(* CODESYS project Brauanlagev3.project

Project tree, tasks and I/O mapping:
  Device : CODESYS Control for Raspberry Pi, 3S - Smart Software Solutions GmbH, version 3.5.9.20
    application Application
      libraries: Standard, * (System); SysProcess, 3.5.7.0 (System); VisuDialogs, * (System); BASIC, 3.3.3.0 (OSCAT); SysTypes Interfaces, * (System); SysMem, 3.5.5.0 (System)
      task VISU_TASK (cyclic, interval 100 ms, priority 31) calls VisuElems.Visu_Prg
      task LinuxSystemTask (cyclic, interval 1000 ms, priority 31) calls RPI_SYSTEM
      task IO (cyclic, interval 10 ms, priority 1) calls IOCOM
      task KI (cyclic, interval 10 ms, priority 1) calls Automatik
      global variables Variablenliste
      visualisation Visualization
      program Automatik [ST]
      visualisation Setup
      visualisation Settings
      program IOCOM [ST]
      program RPI_SYSTEM [ST]
      global variables PersistentVars
    SoftMotion General Axis Pool
    I²C
    SPI
    GPIOs_B_Pi2 : GPIOs B+/Pi2, 3S - Smart Software Solutions GmbH, version 1.1.1.10
        unmapped channels: digital inputs (GPIO0..GPIO31), digital outputs (GPIO0..GPIO31)
    Onewire
      Onewire_master : Onewire master, 3S - Smart Software Solutions GmbH, version 1.0.0.0
        DS18B20 : DS18B20, 3S - Smart Software Solutions GmbH, version 1.3.0.0
            settings: Unique device address = '28-011572667aff'
        DS18B20_2 : DS18B20, 3S - Smart Software Solutions GmbH, version 1.3.0.0
            settings: Unique device address = '28-0115726f14ff'
        DS18B20_1 : DS18B20, 3S - Smart Software Solutions GmbH, version 1.3.0.0
            settings: Unique device address = '28-0115729769ff'
    Camera device
      <Leer>
  libraries: VisuSymbols, 3.5.8.0 (System)
  text list GlobalTextList
  text list System
*)

// Device/Application/Variablenliste
VAR_GLOBAL
	AUTO_VERBLEIBENDE_ZEIT:TIME;
	seek:UINT;
	seek2:UINT;
	IN_TEMP_1:REAL:=0;
	IN_TEMP_2:REAL:=0;
	IN_TEMP_3:REAL:=0;
	OUT_TOPF_2_ON:BOOL:=0;
	OUT_220_1_ON:BOOL:=0;
	OUT_220_2_ON:BOOL:=0;
	OUT_24_1_ON:BOOL:=0;
	OUT_24_2_ON:BOOL:=0;
	OUT_DOSE_1_ON:BOOL:=0;
	OUT_DOSE_2_ON:BOOL:=0;
	OUT_DOSE_3_ON:BOOL:=0;
	OUT_DOSE_4_ON:BOOL:=0;
	OUT_ALARM_ON:BOOL:=0;
END_VAR

{attribute 'qualified_only'}
VAR_GLOBAL PERSISTENT RETAIN
	// Laufzeitvariablen
	AUTO_ZYKLUS:UINT;
	AUTO_REZEPT:UINT;
	AUTO_ON:BOOL;
	// Automatik Rezept
	SET_AUTO_REZEPT_NAME:ARRAY[0..100] OF STRING;
	SET_AUTO_NAME:ARRAY[0..100,0..100] OF STRING;
	SET_AUTO_ZEIT:ARRAY[0..100,0..100] OF UINT;
	SET_AUTO_TIMER_ON:ARRAY[0..100,0..100] OF BOOL;
	SET_AUTO_ALARM:ARRAY[0..100,0..100] OF BOOL;	
	SET_AUTO_TOPF_1_ON:ARRAY[0..100,0..100] OF BOOL;
	SET_AUTO_TOPF_3_ON:ARRAY[0..100,0..100] OF BOOL;
	SET_AUTO_TOPF_1_TARGET:ARRAY[0..100,0..100] OF REAL;
	SET_AUTO_TOPF_3_TARGET:ARRAY[0..100,0..100] OF REAL;
	SET_AUTO_DOSE_1_ON:ARRAY[0..100,0..100] OF BOOL;
	SET_AUTO_DOSE_2_ON:ARRAY[0..100,0..100] OF BOOL;	
	SET_AUTO_DOSE_3_ON:ARRAY[0..100,0..100] OF BOOL;	
	SET_AUTO_DOSE_4_ON:ARRAY[0..100,0..100] OF BOOL;
	// Einstellungen
	SET_TOPF_1_AUTO:BOOL;
	SET_TOPF_3_AUTO:BOOL;
	SET_TOPF_1_TARGET:REAL;
	SET_TOPF_3_TARGET:REAL;
	SET_TOPF_1_HYSTERESIS:REAL:=2;
	SET_TOPF_3_HYSTERESIS:REAL:=2;
	SET_TOPF_1_HYSTERESIS2:REAL:=2;
	SET_TOPF_3_HYSTERESIS2:REAL:=2;
	SET_TOPF_1_ON:BOOL;
	SET_TOPF_3_ON:BOOL;
	SET_TOPF_1_NAME:STRING:='TOPF1';
	SET_TOPF_2_NAME:STRING:='TOPF2';
	SET_TOPF_3_NAME:STRING:='TOPF3';
	SET_DOSE_1_AUTO:BOOL;
	SET_DOSE_2_AUTO:BOOL;
	SET_DOSE_3_AUTO:BOOL;
	SET_DOSE_4_AUTO:BOOL;
	SET_DOSE_1_NAME:STRING:='DOSE1';
	SET_DOSE_2_NAME:STRING:='DOSE2';
	SET_DOSE_3_NAME:STRING:='DOSE3';
	SET_DOSE_4_NAME:STRING:='DOSE4';
END_VAR

// Device/Application/PersistentVars
{attribute 'qualified_only'}
VAR_GLOBAL PERSISTENT RETAIN

	// Instanzpfad der persistenten Variablen erzeugt
	Variablenliste.AUTO_ZYKLUS: UINT;
	// Instanzpfad der persistenten Variablen erzeugt
	Variablenliste.AUTO_REZEPT: UINT;
	// Instanzpfad der persistenten Variablen erzeugt
	Variablenliste.AUTO_ON: BOOL;
	// Instanzpfad der persistenten Variablen erzeugt
	Variablenliste.SET_AUTO_REZEPT_NAME: ARRAY [0..100] OF STRING;
	// Instanzpfad der persistenten Variablen erzeugt
	Variablenliste.SET_AUTO_NAME: ARRAY [0..100, 0..100] OF STRING;
	// Instanzpfad der persistenten Variablen erzeugt
	Variablenliste.SET_AUTO_ZEIT: ARRAY [0..100, 0..100] OF UINT;
	// Instanzpfad der persistenten Variablen erzeugt
	Variablenliste.SET_AUTO_TIMER_ON: ARRAY [0..100, 0..100] OF BOOL;
	// Instanzpfad der persistenten Variablen erzeugt
	Variablenliste.SET_AUTO_ALARM: ARRAY [0..100, 0..100] OF BOOL;
	// Instanzpfad der persistenten Variablen erzeugt
	Variablenliste.SET_AUTO_TOPF_1_ON: ARRAY [0..100, 0..100] OF BOOL;
	// Instanzpfad der persistenten Variablen erzeugt
	Variablenliste.SET_AUTO_TOPF_3_ON: ARRAY [0..100, 0..100] OF BOOL;
	// Instanzpfad der persistenten Variablen erzeugt
	Variablenliste.SET_AUTO_TOPF_1_TARGET: ARRAY [0..100, 0..100] OF REAL;
	// Instanzpfad der persistenten Variablen erzeugt
	Variablenliste.SET_AUTO_TOPF_3_TARGET: ARRAY [0..100, 0..100] OF REAL;
	// Instanzpfad der persistenten Variablen erzeugt
	Variablenliste.SET_AUTO_DOSE_1_ON: ARRAY [0..100, 0..100] OF BOOL;
	// Instanzpfad der persistenten Variablen erzeugt
	Variablenliste.SET_AUTO_DOSE_2_ON: ARRAY [0..100, 0..100] OF BOOL;
	// Instanzpfad der persistenten Variablen erzeugt
	Variablenliste.SET_AUTO_DOSE_3_ON: ARRAY [0..100, 0..100] OF BOOL;
	// Instanzpfad der persistenten Variablen erzeugt
	Variablenliste.SET_AUTO_DOSE_4_ON: ARRAY [0..100, 0..100] OF BOOL;
	// Instanzpfad der persistenten Variablen erzeugt
	Variablenliste.SET_TOPF_1_AUTO: BOOL;
	// Instanzpfad der persistenten Variablen erzeugt
	Variablenliste.SET_TOPF_3_AUTO: BOOL;
	// Instanzpfad der persistenten Variablen erzeugt
	Variablenliste.SET_TOPF_1_TARGET: REAL;
	// Instanzpfad der persistenten Variablen erzeugt
	Variablenliste.SET_TOPF_3_TARGET: REAL;
	// Instanzpfad der persistenten Variablen erzeugt
	Variablenliste.SET_TOPF_1_HYSTERESIS: REAL := 2.0;
	// Instanzpfad der persistenten Variablen erzeugt
	Variablenliste.SET_TOPF_3_HYSTERESIS: REAL := 2.0;
	// Instanzpfad der persistenten Variablen erzeugt
	Variablenliste.SET_TOPF_1_HYSTERESIS2: REAL := 2.0;
	// Instanzpfad der persistenten Variablen erzeugt
	Variablenliste.SET_TOPF_3_HYSTERESIS2: REAL := 2.0;
	// Instanzpfad der persistenten Variablen erzeugt
	Variablenliste.SET_TOPF_1_ON: BOOL;
	// Instanzpfad der persistenten Variablen erzeugt
	Variablenliste.SET_TOPF_3_ON: BOOL;
	// Instanzpfad der persistenten Variablen erzeugt
	Variablenliste.SET_TOPF_1_NAME: STRING := 'TOPF1';
	// Instanzpfad der persistenten Variablen erzeugt
	Variablenliste.SET_TOPF_2_NAME: STRING := 'TOPF2';
	// Instanzpfad der persistenten Variablen erzeugt
	Variablenliste.SET_TOPF_3_NAME: STRING := 'TOPF3';
	// Instanzpfad der persistenten Variablen erzeugt
	Variablenliste.SET_DOSE_1_AUTO: BOOL;
	// Instanzpfad der persistenten Variablen erzeugt
	Variablenliste.SET_DOSE_2_AUTO: BOOL;
	// Instanzpfad der persistenten Variablen erzeugt
	Variablenliste.SET_DOSE_3_AUTO: BOOL;
	// Instanzpfad der persistenten Variablen erzeugt
	Variablenliste.SET_DOSE_4_AUTO: BOOL;
	// Instanzpfad der persistenten Variablen erzeugt
	Variablenliste.SET_DOSE_1_NAME: STRING := 'DOSE1';
	// Instanzpfad der persistenten Variablen erzeugt
	Variablenliste.SET_DOSE_2_NAME: STRING := 'DOSE2';
	// Instanzpfad der persistenten Variablen erzeugt
	Variablenliste.SET_DOSE_3_NAME: STRING := 'DOSE3';
	// Instanzpfad der persistenten Variablen erzeugt
	Variablenliste.SET_DOSE_4_NAME: STRING := 'DOSE4';
END_VAR

// Device/Application/RPI_SYSTEM
PROGRAM RPI_SYSTEM
VAR
   cmdResult   :    RTS_IEC_result;
END_VAR

IF OUT_ALARM_ON THEN 
	// SysProcessExecuteCommand('aplay /media/shared/alarm.wav', ADR(cmdResult)); 
	// SysProcessExecuteCommand('python /media/shared/alarm.py', ADR(cmdResult)); 
END_IF

END_PROGRAM

// Device/Application/IOCOM
PROGRAM IOCOM
VAR
	rTemp: REAL;
END_VAR


%QX0.5:=NOT OUT_DOSE_1_ON;
%QX0.6:=NOT OUT_DOSE_2_ON;
%QX1.4:=NOT OUT_DOSE_3_ON;
%QX1.5:=NOT OUT_DOSE_4_ON;
%QX2.0:=NOT OUT_220_1_ON;
%QX2.3:=NOT OUT_220_2_ON;
%QX2.4:=NOT OUT_24_1_ON;
%QX2.5:=NOT OUT_24_2_ON;
IN_TEMP_1:=DS18B20.rTemp;
IN_TEMP_2:=DS18b20_1.rTemp;
IN_TEMP_3:=DS18b20_2.rTemp;

END_PROGRAM

// Device/Application/Automatik
PROGRAM Automatik
VAR
	TIMER:TON;
END_VAR

(*TODO
ALARM pwm jack`?
*)


TIMER(IN:=SET_AUTO_TIMER_ON[AUTO_ZYKLUS,AUTO_REZEPT] AND AUTO_ON AND NOT TIMER.Q, PT:=LWORD_TO_TIME(UINT_TO_LWORD(SET_AUTO_ZEIT[AUTO_ZYKLUS,AUTO_REZEPT])*60000));
(*TIMER.ET:=ELAPSED;*)
AUTO_VERBLEIBENDE_ZEIT:=LWORD_TO_TIME(UINT_TO_LWORD(SET_AUTO_ZEIT[AUTO_ZYKLUS,AUTO_REZEPT])*60000)-TIMER.ET;


IF TIMER.Q THEN
	AUTO_ZYKLUS:=AUTO_ZYKLUS+1;
	IF SET_AUTO_ALARM[AUTO_ZYKLUS,AUTO_REZEPT] THEN
		OUT_ALARM_ON:=TRUE;
	END_IF
END_IF



IF AUTO_ON THEN
	IF SET_DOSE_1_AUTO THEN
		IF SET_AUTO_DOSE_1_ON[AUTO_ZYKLUS,AUTO_REZEPT] THEN
			OUT_DOSE_1_ON:=TRUE;
		ELSE 
			OUT_DOSE_1_ON:=FALSE;
		END_IF
	END_IF
	
	IF SET_DOSE_2_AUTO THEN
		IF SET_AUTO_DOSE_2_ON[AUTO_ZYKLUS,AUTO_REZEPT] THEN
			OUT_DOSE_2_ON:=TRUE;
		ELSE 
			OUT_DOSE_2_ON:=FALSE;
		END_IF
	END_IF

	IF SET_DOSE_3_AUTO THEN
		IF SET_AUTO_DOSE_3_ON[AUTO_ZYKLUS,AUTO_REZEPT] THEN
			OUT_DOSE_3_ON:=TRUE;
		ELSE 
			OUT_DOSE_3_ON:=FALSE;
		END_IF
	END_IF

	IF SET_DOSE_4_AUTO THEN
		IF SET_AUTO_DOSE_4_ON[AUTO_ZYKLUS,AUTO_REZEPT] THEN
			OUT_DOSE_4_ON:=TRUE;
		ELSE 
			OUT_DOSE_4_ON:=FALSE;
		END_IF
	END_IF

	IF SET_TOPF_1_AUTO THEN
		IF SET_AUTO_TOPF_1_ON[AUTO_ZYKLUS,AUTO_REZEPT] THEN
			SET_TOPF_1_TARGET:=SET_AUTO_TOPF_1_TARGET[AUTO_ZYKLUS,AUTO_REZEPT];
			SET_TOPF_1_ON:=TRUE;
		ELSE
			SET_TOPF_1_ON:=FALSE;
		END_IF
	END_IF

	IF SET_TOPF_3_AUTO THEN
		IF SET_AUTO_TOPF_3_ON[AUTO_ZYKLUS,AUTO_REZEPT] THEN
			SET_TOPF_3_TARGET:=SET_AUTO_TOPF_3_TARGET[AUTO_ZYKLUS,AUTO_REZEPT];
			SET_TOPF_3_ON:=TRUE;
		ELSE
			SET_TOPF_3_ON:=FALSE;
		END_IF
	END_IF
END_IF

IF SET_TOPF_1_ON THEN
	IF IN_TEMP_1 > SET_TOPF_1_TARGET THEN
		OUT_220_1_ON:=FALSE;
		OUT_24_1_ON:=FALSE;
	END_IF
	IF IN_TEMP_1 < SET_TOPF_1_TARGET - SET_TOPF_1_HYSTERESIS THEN
		OUT_220_1_ON:=TRUE;
	END_IF
	IF IN_TEMP_1 < SET_TOPF_1_TARGET - SET_TOPF_1_HYSTERESIS - SET_TOPF_1_HYSTERESIS2 THEN
		OUT_24_1_ON:=TRUE;
	ELSE
		OUT_24_1_ON:=FALSE;
	END_IF
ELSE 
	OUT_220_1_ON:=FALSE;
	OUT_24_1_ON:=FALSE;
END_IF

IF SET_TOPF_3_ON THEN
	IF IN_TEMP_3 > SET_TOPF_3_TARGET THEN
		OUT_220_2_ON:=FALSE;
		OUT_24_2_ON:=FALSE;
	END_IF
	IF IN_TEMP_3 < SET_TOPF_3_TARGET - SET_TOPF_3_HYSTERESIS THEN
		OUT_220_2_ON:=TRUE;
	END_IF
	IF IN_TEMP_3 < SET_TOPF_3_TARGET - SET_TOPF_3_HYSTERESIS - SET_TOPF_3_HYSTERESIS2 THEN
		OUT_24_2_ON:=TRUE;
	ELSE
		OUT_24_2_ON:=FALSE;
	END_IF
ELSE 
	OUT_220_2_ON:=FALSE;
	OUT_24_2_ON:=FALSE;
END_IF

END_PROGRAM

// Device/Application/Visualization
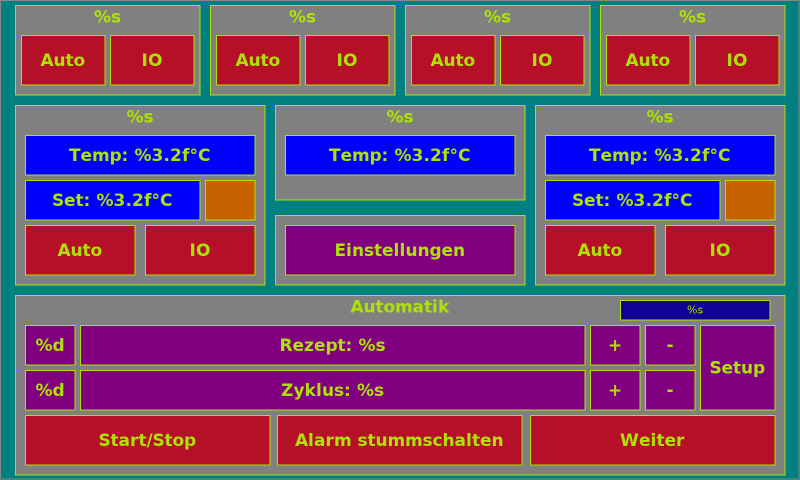
VISUALIZATION Visualization  // 800x480
    RoundedRectangle (15,295 770x180), "Automatik"
    RoundedRectangle (25,415 245x50), "Start/Stop", colour toggle: AUTO_ON
        toggle AUTO_ON
    RoundedRectangle (277,415 245x50), "Alarm stummschalten", colour toggle: OUT_ALARM_ON
        OnMouseDown: execute { OUT_ALARM_ON:=0; }
    RoundedRectangle (700,325 75x85), "Setup"
        OnMouseDown:  Assign=Setup, Type=Assignment
    RoundedRectangle (530,415 245x50), "Weiter"
        OnMouseDown: execute { AUTO_ZYKLUS:=AUTO_ZYKLUS+1; }
    RoundedRectangle (15,5 185x90), "%s", text variable: SET_DOSE_1_NAME
        OnMouseDown: write the text variable via Edit
    RoundedRectangle (110,35 84x50), "IO", colour toggle: OUT_DOSE_1_ON
        toggle OUT_DOSE_1_ON
    RoundedRectangle (21,35 84x50), "Auto", colour toggle: SET_DOSE_1_AUTO
        toggle SET_DOSE_1_AUTO
    RoundedRectangle (210,5 185x90), "%s", text variable: SET_DOSE_2_NAME
        OnMouseDown: write the text variable via Edit
    RoundedRectangle (305,35 84x50), "IO", colour toggle: OUT_DOSE_2_ON
        toggle OUT_DOSE_2_ON
    RoundedRectangle (216,35 84x50), "Auto", colour toggle: SET_DOSE_2_AUTO
        toggle SET_DOSE_2_AUTO
    RoundedRectangle (405,5 185x90), "%s", text variable: SET_DOSE_3_NAME
        OnMouseDown: write the text variable via Edit
    RoundedRectangle (500,35 84x50), "IO", colour toggle: OUT_DOSE_3_ON
        toggle OUT_DOSE_3_ON
    RoundedRectangle (411,35 84x50), "Auto", colour toggle: SET_DOSE_3_AUTO
        toggle SET_DOSE_3_AUTO
    RoundedRectangle (600,5 185x90), "%s", text variable: SET_DOSE_4_NAME
        OnMouseDown: write the text variable via Edit
    RoundedRectangle (695,35 84x50), "IO", colour toggle: OUT_DOSE_4_ON
        toggle OUT_DOSE_4_ON
    RoundedRectangle (606,35 84x50), "Auto", colour toggle: SET_DOSE_4_AUTO
        toggle SET_DOSE_4_AUTO
    RoundedRectangle (275,105 250x95), "%s", text variable: SET_TOPF_2_NAME
        OnMouseDown: write the text variable via Edit
    RoundedRectangle (285,135 230x40), "Temp: %3.2f°C", text variable: IN_TEMP_2
    RoundedRectangle (535,105 250x180), "%s", text variable: SET_TOPF_3_NAME, colour toggle: OUT_220_2_ON
        OnMouseDown: write the text variable via Edit
    RoundedRectangle (665,225 110x50), "IO", colour toggle: SET_TOPF_3_ON
        toggle SET_TOPF_3_ON
    RoundedRectangle (545,225 110x50), "Auto", colour toggle: SET_TOPF_3_AUTO
        toggle SET_TOPF_3_AUTO
    RoundedRectangle (545,135 230x40), "Temp: %3.2f°C", text variable: IN_TEMP_3
    RoundedRectangle (545,180 175x40), "Set: %3.2f°C", text variable: SET_TOPF_3_TARGET
        OnMouseDown: write the text variable via Edit, min 0, max 105
    RoundedRectangle (725,180 50x40), text variable: SET_TOPF_3_TARGET
        OnMouseDown: write the text variable via VisuDialogs.Numpad, min 0, max 105
    RoundedRectangle (15,105 250x180), "%s", text variable: SET_TOPF_1_NAME, colour toggle: OUT_220_1_ON
        OnMouseDown: write the text variable via Edit
    RoundedRectangle (145,225 110x50), "IO", colour toggle: SET_TOPF_1_ON
        toggle SET_TOPF_1_ON
    RoundedRectangle (25,225 110x50), "Auto", colour toggle: SET_TOPF_1_AUTO
        toggle SET_TOPF_1_AUTO
    RoundedRectangle (25,135 230x40), "Temp: %3.2f°C", text variable: IN_TEMP_1
    RoundedRectangle (25,180 175x40), "Set: %3.2f°C", text variable: SET_TOPF_1_TARGET
        OnMouseDown: write the text variable via Edit, min 0, max 105
    RoundedRectangle (205,180 50x40), text variable: SET_TOPF_1_TARGET
        OnMouseDown: write the text variable via VisuDialogs.Numpad, min 0, max 105
    RoundedRectangle (275,215 250x70)
    RoundedRectangle (285,225 230x50), "Einstellungen"
        OnMouseDown:  Assign=Settings, Type=Assignment
    RoundedRectangle (620,300 150x20), "%s", text variable: AUTO_VERBLEIBENDE_ZEIT, invisible if: NOT SET_AUTO_TIMER_ON[AUTO_ZYKLUS,AUTO_REZEPT]
    RoundedRectangle (590,370 50x40), "+"
        OnMouseDown: execute { AUTO_ZYKLUS:=AUTO_ZYKLUS+1; }
    RoundedRectangle (645,370 50x40), "-"
        OnMouseDown: execute {
            IF AUTO_ZYKLUS > 0 THEN
            	AUTO_ZYKLUS:=AUTO_ZYKLUS-1;
            END_IF;
        }
    RoundedRectangle (80,370 505x40), "Zyklus: %s", text variable: SET_AUTO_NAME[AUTO_ZYKLUS,AUTO_REZEPT]
    RoundedRectangle (25,370 50x40), "%d", text variable: AUTO_ZYKLUS
    RoundedRectangle (590,325 50x40), "+"
        OnMouseDown: execute { AUTO_REZEPT:=AUTO_REZEPT+1; AUTO_ON:=FALSE; }
    RoundedRectangle (645,325 50x40), "-"
        OnMouseDown: execute {
            IF AUTO_REZEPT > 0 THEN
            	AUTO_REZEPT:=AUTO_REZEPT-1;
            END_IF;
            AUTO_ON:=FALSE;
        }
    RoundedRectangle (80,325 505x40), "Rezept: %s", text variable: SET_AUTO_REZEPT_NAME[AUTO_REZEPT]
    RoundedRectangle (25,325 50x40), "%d", text variable: AUTO_REZEPT
END_VISUALIZATION

// Device/Application/Setup
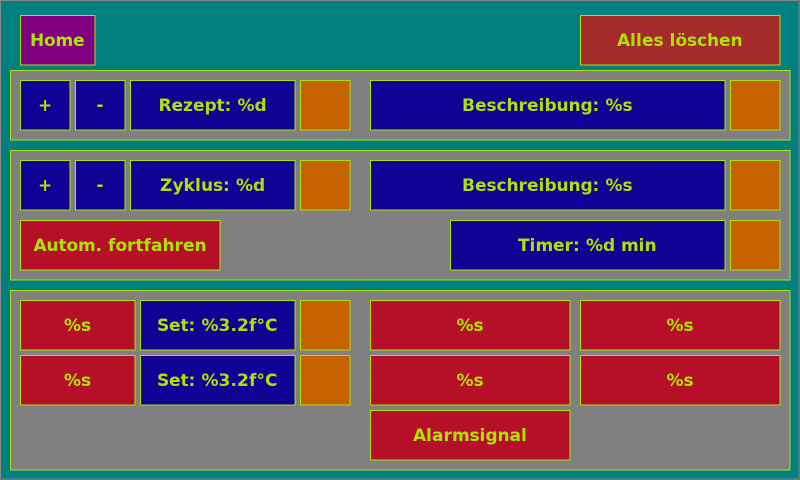
VISUALIZATION Setup  // 800x480
    RoundedRectangle (10,70 780x70)
    RoundedRectangle (10,290 780x180)
    RoundedRectangle (10,150 780x130)
    RoundedRectangle (20,300 115x50), "%s", text variable: SET_TOPF_1_NAME, colour toggle: SET_AUTO_TOPF_1_ON[seek,seek2]
        toggle SET_AUTO_TOPF_1_ON[seek,seek2]
    RoundedRectangle (140,300 155x50), "Set: %3.2f°C", text variable: SET_AUTO_TOPF_1_TARGET[seek,seek2]
        OnMouseDown: write the text variable via Edit
    RoundedRectangle (300,300 50x50), text variable: SET_AUTO_TOPF_1_TARGET[seek,seek2]
        OnMouseDown: write the text variable via VisuDialogs.Numpad
    RoundedRectangle (370,300 200x50), "%s", text variable: SET_DOSE_1_NAME, colour toggle: SET_AUTO_DOSE_1_ON[seek,seek2]
        toggle SET_AUTO_DOSE_1_ON[seek,seek2]
    RoundedRectangle (370,410 200x50), "Alarmsignal", colour toggle: SET_AUTO_ALARM[seek,seek2]
        toggle SET_AUTO_ALARM[seek,seek2]
    RoundedRectangle (20,355 115x50), "%s", text variable: SET_TOPF_3_NAME, colour toggle: SET_AUTO_TOPF_3_ON[seek,seek2]
        toggle SET_AUTO_TOPF_3_ON[seek,seek2]
    RoundedRectangle (300,355 50x50), text variable: SET_AUTO_TOPF_3_TARGET[seek,seek2]
        OnMouseDown: write the text variable via VisuDialogs.Numpad
    RoundedRectangle (140,355 155x50), "Set: %3.2f°C", text variable: SET_AUTO_TOPF_3_TARGET[seek,seek2]
        OnMouseDown: write the text variable via Edit
    RoundedRectangle (370,355 200x50), "%s", text variable: SET_DOSE_2_NAME, colour toggle: SET_AUTO_DOSE_2_ON[seek,seek2]
        toggle SET_AUTO_DOSE_2_ON[seek,seek2]
    RoundedRectangle (580,355 200x50), "%s", text variable: SET_DOSE_4_NAME, colour toggle: SET_AUTO_DOSE_4_ON[seek,seek2]
        toggle SET_AUTO_DOSE_4_ON[seek,seek2]
    RoundedRectangle (580,300 200x50), "%s", text variable: SET_DOSE_3_NAME, colour toggle: SET_AUTO_DOSE_3_ON[seek,seek2]
        toggle SET_AUTO_DOSE_3_ON[seek,seek2]
    RoundedRectangle (20,15 75x50), "Home"
        OnMouseDown:  Assign=Visualization, Type=Assignment
    RoundedRectangle (370,160 355x50), "Beschreibung: %s", text variable: SET_AUTO_NAME[seek,seek2]
        OnMouseDown: write the text variable via Edit
    RoundedRectangle (730,160 50x50), text variable: SET_AUTO_NAME[seek,seek2]
        OnMouseDown: write the text variable via VisuDialogs.Keypad
    RoundedRectangle (20,160 50x50), "+"
        OnMouseDown: execute { seek:=seek+1; }
    RoundedRectangle (75,160 50x50), "-"
        OnMouseDown: execute {
            IF seek > 0 THEN
            	seek:=seek-1;
            END_IF;
        }
    RoundedRectangle (130,160 165x50), "Zyklus: %d", text variable: seek
        OnMouseDown: write the text variable via Edit
    RoundedRectangle (300,160 50x50), text variable: seek
        OnMouseDown: write the text variable via VisuDialogs.Numpad
    RoundedRectangle (450,220 275x50), "Timer: %d min", text variable: SET_AUTO_ZEIT[seek,seek2], invisible if: NOT SET_AUTO_TIMER_ON[seek,seek2]
        OnMouseDown: write the text variable via Edit
    RoundedRectangle (730,220 50x50), text variable: SET_AUTO_ZEIT[seek,seek2], invisible if: NOT SET_AUTO_TIMER_ON[seek,seek2]
        OnMouseDown: write the text variable via VisuDialogs.Numpad
    RoundedRectangle (20,220 200x50), "Autom. fortfahren", colour toggle: SET_AUTO_TIMER_ON[seek,seek2]
        toggle SET_AUTO_TIMER_ON[seek,seek2]
    RoundedRectangle (580,15 200x50), "Alles löschen"
        OnMouseDown: execute {
            SysMemSet(pDest:=ADR(SET_AUTO_NAME) , udiValue:= 0, udiCount:= SIZEOF(SET_AUTO_NAME));
            SysMemSet(pDest:=ADR(SET_AUTO_ZEIT) , udiValue:= 0, udiCount:= SIZEOF(SET_AUTO_ZEIT));
            SysMemSet(pDest:=ADR(SET_AUTO_TIMER_ON) , udiValue:= 0, udiCount:= SIZEOF(SET_AUTO_TIMER_ON));
            SysMemSet(pDest:=ADR(SET_AUTO_ALARM) , udiValue:= 0, udiCount:= SIZEOF(SET_AUTO_ALARM));
            SysMemSet(pDest:=ADR(SET_AUTO_TOPF_1_ON) , udiValue:= 0, udiCount:= SIZEOF(SET_AUTO_TOPF_1_ON));
            SysMemSet(pDest:=ADR(SET_AUTO_TOPF_3_ON) , udiValue:= 0, udiCount:= SIZEOF(SET_AUTO_TOPF_3_ON));
            SysMemSet(pDest:=ADR(SET_AUTO_TOPF_1_TARGET) , udiValue:= 0, udiCount:= SIZEOF(SET_AUTO_TOPF_1_TARGET));
            SysMemSet(pDest:=ADR(SET_AUTO_TOPF_3_TARGET) , udiValue:= 0, udiCount:= SIZEOF(SET_AUTO_TOPF_3_TARGET));
            SysMemSet(pDest:=ADR(SET_AUTO_DOSE_1_ON) , udiValue:= 0, udiCount:= SIZEOF(SET_AUTO_DOSE_1_ON));
            SysMemSet(pDest:=ADR(SET_AUTO_DOSE_2_ON) , udiValue:= 0, udiCount:= SIZEOF(SET_AUTO_DOSE_2_ON));
            SysMemSet(pDest:=ADR(SET_AUTO_DOSE_3_ON) , udiValue:= 0, udiCount:= SIZEOF(SET_AUTO_DOSE_3_ON));
            SysMemSet(pDest:=ADR(SET_AUTO_DOSE_4_ON) , udiValue:= 0, udiCount:= SIZEOF(SET_AUTO_DOSE_4_ON));
            SysMemSet(pDest:=ADR(SET_AUTO_REZEPT_NAME) , udiValue:= 0, udiCount:= SIZEOF(SET_AUTO_REZEPT_NAME));
        }
    RoundedRectangle (20,80 50x50), "+"
        OnMouseDown: execute { seek2:=seek2+1; }
    RoundedRectangle (75,80 50x50), "-"
        OnMouseDown: execute {
            IF seek2 > 0 THEN
            	seek2:=seek2-1;
            END_IF;
        }
    RoundedRectangle (130,80 165x50), "Rezept: %d", text variable: seek2
        OnMouseDown: write the text variable via Edit
    RoundedRectangle (300,80 50x50), text variable: seek2
        OnMouseDown: write the text variable via VisuDialogs.Numpad
    RoundedRectangle (370,80 355x50), "Beschreibung: %s", text variable: SET_AUTO_REZEPT_NAME[seek2]
        OnMouseDown: write the text variable via Edit
    RoundedRectangle (730,80 50x50), text variable: SET_AUTO_REZEPT_NAME[seek2]
        OnMouseDown: write the text variable via VisuDialogs.Keypad
END_VISUALIZATION

// Device/Application/Settings
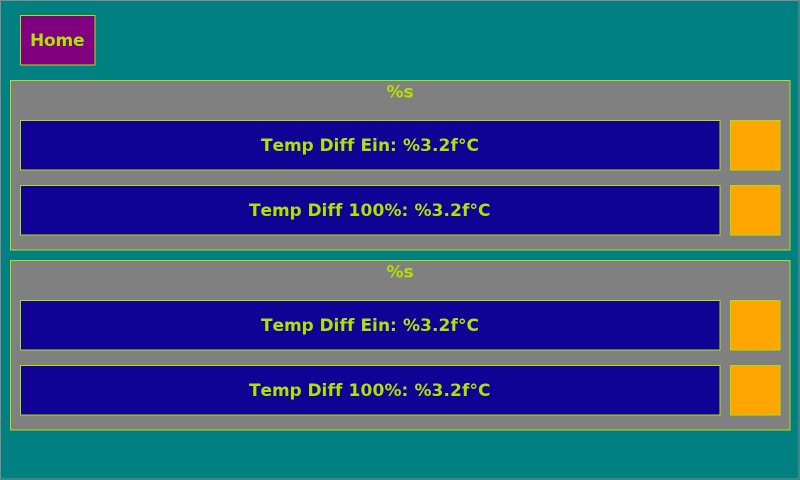
VISUALIZATION Settings  // 800x480
    RoundedRectangle (10,260 780x170), "%s", text variable: SET_TOPF_3_NAME
        OnMouseDown: write the text variable via Edit
    RoundedRectangle (10,80 780x170), "%s", text variable: SET_TOPF_1_NAME
        OnMouseDown: write the text variable via Edit
    RoundedRectangle (20,15 75x50), "Home"
        OnMouseDown:  Assign=Visualization, Type=Assignment
    RoundedRectangle (20,120 700x50), "Temp Diff Ein: %3.2f°C", text variable: SET_TOPF_1_HYSTERESIS
        OnMouseDown: write the text variable via Edit
    RoundedRectangle (730,120 50x50), text variable: SET_TOPF_1_HYSTERESIS
        OnMouseDown: write the text variable via VisuDialogs.Numpad
    RoundedRectangle (20,185 700x50), "Temp Diff 100%: %3.2f°C", text variable: SET_TOPF_1_HYSTERESIS2
        OnMouseDown: write the text variable via Edit
    RoundedRectangle (730,185 50x50), text variable: SET_TOPF_1_HYSTERESIS2
        OnMouseDown: write the text variable via VisuDialogs.Numpad
    RoundedRectangle (20,300 700x50), "Temp Diff Ein: %3.2f°C", text variable: SET_TOPF_3_HYSTERESIS
        OnMouseDown: write the text variable via Edit
    RoundedRectangle (730,300 50x50), text variable: SET_TOPF_3_HYSTERESIS
        OnMouseDown: write the text variable via VisuDialogs.Numpad
    RoundedRectangle (20,365 700x50), "Temp Diff 100%: %3.2f°C", text variable: SET_TOPF_3_HYSTERESIS2
        OnMouseDown: write the text variable via Edit
    RoundedRectangle (730,365 50x50), text variable: SET_TOPF_3_HYSTERESIS2
        OnMouseDown: write the text variable via VisuDialogs.Numpad
END_VISUALIZATION

(* text list System (id | default)
  Apr | Apr
  April | April
  Aug | Aug
  August | August
  Dec | Dec
  December | December
  Feb | Feb
  February | February
  Fri | Fri
  Friday | Friday
  Jan | Jan
  January | January
  Jul | Jul
  July | July
  Jun | Jun
  June | June
  Mar | Mar
  March | March
  May | May
  May_3Letter | May
  Mon | Mon
  Monday | Monday
  Nov | Nov
  November | November
  Oct | Oct
  October | October
  Sat | Sat
  Saturday | Saturday
  Sep | Sep
  September | September
  Sun | Sun
  Sunday | Sunday
  Thu | Thu
  Thursday | Thursday
  Tue | Tue
  Tuesday | Tuesday
  Wed | Wed
  Wednesday | Wednesday
   |  *)
